# B&R Automation Studio project cnc
Automation Studio 4.3.6.57 SP; technology packages: Acp10Arnc0 5.2.1, mapp 5.2.1

## Configuration X20CP1382SM

CPU X20CP1382, AutomationRuntime G4.34, Build 4.1.2, Vc V4.34.2

### Task classes (Cpu.sw)
```
Cyclic#1 (cycle 4000 us, tolerance 0 us):
  ncsdcctrl <- Motion.Stepper.ncsdcctrl.prg
Cyclic#3:
  Cnc <- Motion.Cnc.prg
  MFunc <- Motion.MFunc.prg
Cyclic#4:
  Draw <- Visualization.Draw.prg
DataObjects: Acp10sys, Arnc0sys
NcDataObjects: CncInit <- Motion.CncInit.dob, gmcipvar <- GmcIpUserConfig.gmcipvar.dob, gmcipfun <- GmcIpUserConfig.gmcipfun.dob, gmcipfub <- GmcIpUserConfig.gmcipfub.dob, gmcipubr <- GmcIpUserConfig.gmcipubr.dob, gmcipusm <- GmcIpUserConfig.gmcipusm.dob, gmcipui <- GmcIpUserConfig.gmcipui.dob, gmcipus <- GmcIpUserConfig.gmcipus.dob, gmcipuc <- GmcIpUserConfig.gmcipuc.dob, gmcipsys <- GmcIpConfig.gmcipsys.dob, gmciplbr <- GmcIpConfig.gmciplbr.dob, gmcipcbr <- GmcIpConfig.gmcipcbr.dob, gmciplsm <- GmcIpConfig.gmciplsm.dob, gmcipcsm <- GmcIpConfig.gmcipcsm.dob, gmcipcfg <- GmcIpConfig.gmcipcfg.dob, gmcipiec <- GmcIpConfig.gmcipiec.dob, gmciplog <- GmcIpConfig.gmciplog.dob, gmcipesm <- GmcIpConfig.gmcipesm.dob, gmcipmxd <- GmcIpConfig.gmcipmxd.dob, gmcipmx <- GmcIpConfig.gmcipmx.dob, gAxisXa <- Motion.Stepper.gAxisXobj.gAxisXa.dob, gAxisXi <- Motion.Stepper.gAxisXobj.gAxisXi.dob, gAxisYa <- Motion.Stepper.gAxisYobj.gAxisYa.dob, gAxisYi <- Motion.Stepper.gAxisYobj.gAxisYi.dob, acp10etxen <- Motion.acp10etxen.dob, gAxisAa <- Motion.Stepper.gAxisAobj.gAxisAa.dob, gAxisAi <- Motion.Stepper.gAxisAobj.gAxisAi.dob, Micky <- Motion.Micky.dob
VcDataObjects: Visu <- Visualization.Visu.dob
Binaries: TCData, udbdef, arsvcreg, ashwac, Config_4, Config_3, ashwd, Config_1, User, sysconf, asfw, arconfig, iomap, Role, Config, Acp10map, acp10cfg, Arnc0map, arnc0cfg, vcclbox, vcnet, Visu02, vccpopup, vccscale, Visu01, vccddbox, Visu03, vccshape, vcpkat, vctcal, vcmgr, vcpdvnc, vccline, vccovl, vcdsint, vcctext, vccslider, vcrt, vccurl, vcxml, vcshared, vccbmp, vcchspot, vcchtml, vcpdsw, vccdt, vcdsloc, vcalarm, arial, vccalarm, vccstr, vcbclass, vcgclass, vcfntttf, vccnum, vcfile, arialbd, vccbtn, vcpfx20, Config_2, vcctrend, Visu102, Visu103, vccbar, vcpfar00
Libraries: Acp10man, Acp10par, NcGlobal, MpFile, Acp10_MC, brsystem, sys_lib, runtime, Acp10sim, MpCom, MpAxis, Arnc0man, DataObj, AsArLog, FileIO, AsArProf, AsMem, astime, MpCnc, GmcArncGrp, GmcManager, MpWebXs, AsArSdm, Acp10sdc, MpAlarmX, AsBrStr, MpBase, GmcGrpAPI, asieccon, powerlnk, areventlog, vcresman, arsvcreg, ashw, visapi
```

### Hardware
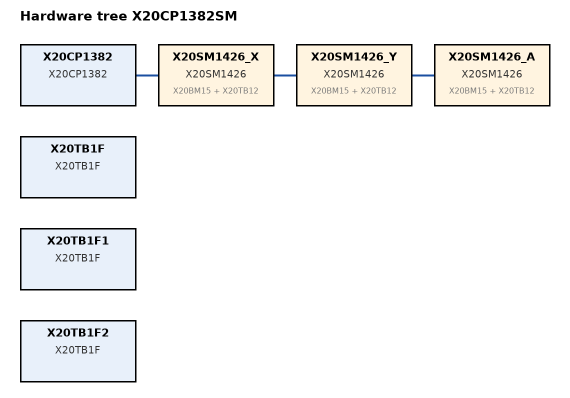
```
X20BM15 : X20BM15 v1.0.1.0  [X2X1 -> X20CP1382.IF6 (NodeNumber=1)]
X20BM15a : X20BM15 v1.0.1.0  [X2X1 -> X20BM15.X2X2 (NodeNumber=2)]
X20BM15b : X20BM15 v1.0.1.0  [X2X1 -> X20BM15a.X2X2 (NodeNumber=3)]
X20CP1382 : X20CP1382 v1.6.1.0  [X1 -> X1.SL; X2 -> X2.SL; X3 -> X3.SL]
  Module X1 (Type=X1, Virtual=true, Version=1.6.1.0)
    Connection (Connector=SS1, TargetModule=X20TB1F, TargetConnector=SS)
    Connection (Connector=SL, TargetModule=X20CP1382, TargetConnector=X1)
  Module X2 (Type=X2, Virtual=true, Version=1.6.1.0)
    Connection (Connector=SS1, TargetModule=X20TB1F1, TargetConnector=SS)
    Connection (Connector=SL, TargetModule=X20CP1382, TargetConnector=X2)
  Module X3 (Type=X3, Virtual=true, Version=1.6.1.0)
    Connection (Connector=SS1, TargetModule=X20TB1F2, TargetConnector=SS)
    Connection (Connector=SL, TargetModule=X20CP1382, TargetConnector=X3)
  Connector IF2:
    ActivateDevice = 1
    Mode = Manual
    InternetAddress = 192.168.0.1
    SubnetMask = 255.255.255.0
    InaNodeNumber = 0
    Vnc1
    VncVcObjectName1 = Visu
    VncKeyMappingFile1 = VC\PS2-Keyboard.dis
    VncRefreshRate1 = 200
  Connector IF3:
    CycleTime = 2000
  ConfigurationID = cnc_X20CP1382SM
  UserPartitionSize = 500
  Simulation = 1
  TimerDeviceType = EPLX2X
  TimerDevice = X20CP1382.IF3
  TaskClassIdleTime = 4000
  Cyclic1Duration = 4000
  Cyclic1Tolerance = 0
  FileDevice1
  FileDeviceName1 = CNC_PrgDir
  FileDevicePath1 = F:\CNC_PrgDir\
  FtpUser1
  FtpUsername1 = ich
  FtpUserPassword1 = 0jkekh+UYz/SowwWBzua0G3yXD3GBpeVHnITZJiG9J0=
  FtpUserSalt1 = 4HMg2Zqv
  FTPAccessRight1 = 0
X20SM1426_A : X20SM1426 v1.5.1.1  [SS1 -> X20TB12b.SS; SL -> X20BM15b.SL1]
  Supervision = off
  RatedCurrent = 50
  MaximumCurrent = 50
  LatchSync = Stepper latch value synchron (AB/R latch value asynchron)
  SM_SCALE_LOAD_UNITS_r1 = 36000
  SCALE_ENCOD_INCR_r1 = 51200
  CNC_r1 = on
  BothEndSwitchesAreNormallyOpen_r1 = on
  QuickStopIsNormallyOpen_r1 = on
X20SM1426_X : X20SM1426 v1.5.1.1  [SS1 -> X20TB12.SS; SL -> X20BM15.SL1]
  Supervision = off
  RatedCurrent = 50
  MaximumCurrent = 50
  LatchSync = Stepper latch value synchron (AB/R latch value asynchron)
  SM_SCALE_LOAD_UNITS_r1 = 200
  SCALE_ENCOD_INCR_r1 = 51200
  CNC_r1 = on
  BothEndSwitchesAreNormallyOpen_r1 = on
  QuickStopIsNormallyOpen_r1 = on
X20SM1426_Y : X20SM1426 v1.5.1.1  [SS1 -> X20TB12a.SS; SL -> X20BM15a.SL1]
  Supervision = off
  RatedCurrent = 50
  MaximumCurrent = 50
  LatchSync = Stepper latch value synchron (AB/R latch value asynchron)
  SM_SCALE_LOAD_UNITS_r1 = 200
  SCALE_ENCOD_INCR_r1 = 51200
  CNC_r1 = on
  BothEndSwitchesAreNormallyOpen_r1 = on
  QuickStopIsNormallyOpen_r1 = on
X20TB12 : X20TB12 v1.0.0.0
X20TB12a : X20TB12 v1.0.0.0
X20TB12b : X20TB12 v1.0.0.0
X20TB1F : X20TB1F v1.0.0.0
X20TB1F1 : X20TB1F v1.0.0.0
X20TB1F2 : X20TB1F v1.0.0.0
```

### IoMap.iom - X20CP1382/IoMap.iom
```iecst
VAR_CONFIG
	Cyclic#1.gAxisX_DrvIf.iLifeCnt AT %IB."X20SM1426_X".LifeCnt;
	Cyclic#1.gAxisX_DrvIf.iDrvOK AT %IX."X20SM1426_X".DrvOk01;
	Cyclic#1.gAxisX_DrvIf.oBoostCurrent AT %QX."X20SM1426_X".BoostCurrent01;
	Cyclic#1.gAxisX_DrvIf.oStandStillCurrent AT %QX."X20SM1426_X".StandstillCurrent01;
	Cyclic#1.gAxisX_DrvIf.oSetTime AT %QW."X20SM1426_X".SetTime01;
	Cyclic#1.gAxisX_MotorStep0 AT %QW."X20SM1426_X".Motor1Step0;
	Cyclic#1.gAxisX_DiDoIf.iLifeCntDriveEnable AT %IB."X20SM1426_X".LifeCnt;
	Cyclic#1.gAxisX_DiDoIf.iLifeCntDriveReady AT %IB."X20SM1426_X".LifeCnt;
	Cyclic#1.gAxisX_DiDoIf.iDriveReady AT %IX."X20SM1426_X".DrvOk01;
	Cyclic#1.gAxisX_DiDoIf.oDriveEnable AT %QX."X20SM1426_X".DriveEnable01;
	Cyclic#1.gAxisX_EncIf1.iLifeCnt AT %IB."X20SM1426_X".LifeCnt;
	Cyclic#1.gAxisX_EncIf1.iEncOK AT %IX."X20SM1426_X".EncOk01;
	Cyclic#1.gAxisX_EncIf1.iActPos AT %IW."X20SM1426_X".ActPos01;
	Cyclic#1.gAxisX_EncIf1.iRefPulsePos AT %IW."X20SM1426_X".RefPulsePos01;
	Cyclic#1.gAxisX_EncIf1.iRefPulseCnt AT %IB."X20SM1426_X".RefPulseCnt01;
	Cyclic#1.gAxisX_EncIf1.iActTime AT %IW."X20SM1426_X".ActTime01;
	Cyclic#1.gAxisY_DrvIf.iLifeCnt AT %IB."X20SM1426_Y".LifeCnt;
	Cyclic#1.gAxisY_DrvIf.iDrvOK AT %IX."X20SM1426_Y".DrvOk01;
	Cyclic#1.gAxisY_DrvIf.oBoostCurrent AT %QX."X20SM1426_Y".BoostCurrent01;
	Cyclic#1.gAxisY_DrvIf.oStandStillCurrent AT %QX."X20SM1426_Y".StandstillCurrent01;
	Cyclic#1.gAxisY_DrvIf.oSetTime AT %QW."X20SM1426_Y".SetTime01;
	Cyclic#1.gAxisY_MotorStep0 AT %QW."X20SM1426_Y".Motor1Step0;
	Cyclic#1.gAxisY_DiDoIf.iLifeCntDriveEnable AT %IB."X20SM1426_Y".LifeCnt;
	Cyclic#1.gAxisY_DiDoIf.iLifeCntDriveReady AT %IB."X20SM1426_Y".LifeCnt;
	Cyclic#1.gAxisY_DiDoIf.iDriveReady AT %IX."X20SM1426_Y".DrvOk01;
	Cyclic#1.gAxisY_DiDoIf.oDriveEnable AT %QX."X20SM1426_Y".DriveEnable01;
	Cyclic#1.gAxisY_EncIf1.iLifeCnt AT %IB."X20SM1426_Y".LifeCnt;
	Cyclic#1.gAxisY_EncIf1.iEncOK AT %IX."X20SM1426_Y".EncOk01;
	Cyclic#1.gAxisY_EncIf1.iActPos AT %IW."X20SM1426_Y".ActPos01;
	Cyclic#1.gAxisY_EncIf1.iRefPulsePos AT %IW."X20SM1426_Y".RefPulsePos01;
	Cyclic#1.gAxisY_EncIf1.iRefPulseCnt AT %IB."X20SM1426_Y".RefPulseCnt01;
	Cyclic#1.gAxisY_EncIf1.iActTime AT %IW."X20SM1426_Y".ActTime01;
	Cyclic#1.gAxisA_DrvIf.iLifeCnt AT %IB."X20SM1426_A".LifeCnt;
	Cyclic#1.gAxisA_DrvIf.iDrvOK AT %IX."X20SM1426_A".DrvOk01;
	Cyclic#1.gAxisA_DrvIf.oBoostCurrent AT %QX."X20SM1426_A".BoostCurrent01;
	Cyclic#1.gAxisA_DrvIf.oStandStillCurrent AT %QX."X20SM1426_A".StandstillCurrent01;
	Cyclic#1.gAxisA_DrvIf.oSetTime AT %QW."X20SM1426_A".SetTime01;
	Cyclic#1.gAxisA_MotorStep0 AT %QW."X20SM1426_A".Motor1Step0;
	Cyclic#1.gAxisA_DiDoIf.iLifeCntDriveEnable AT %IB."X20SM1426_A".LifeCnt;
	Cyclic#1.gAxisA_DiDoIf.iLifeCntDriveReady AT %IB."X20SM1426_A".LifeCnt;
	Cyclic#1.gAxisA_DiDoIf.iDriveReady AT %IX."X20SM1426_A".DrvOk01;
	Cyclic#1.gAxisA_DiDoIf.oDriveEnable AT %QX."X20SM1426_A".DriveEnable01;
	Cyclic#1.gAxisA_EncIf1.iLifeCnt AT %IB."X20SM1426_A".LifeCnt;
	Cyclic#1.gAxisA_EncIf1.iEncOK AT %IX."X20SM1426_A".EncOk01;
	Cyclic#1.gAxisA_EncIf1.iActPos AT %IW."X20SM1426_A".ActPos01;
	Cyclic#1.gAxisA_EncIf1.iRefPulsePos AT %IW."X20SM1426_A".RefPulsePos01;
	Cyclic#1.gAxisA_EncIf1.iRefPulseCnt AT %IB."X20SM1426_A".RefPulseCnt01;
	Cyclic#1.gAxisA_EncIf1.iActTime AT %IW."X20SM1426_A".ActTime01;
END_VAR
```

### Acp10cfg.ncc - X20CP1382/Motion/Acp10cfg.ncc
```
NcConfiguration (Version=3.12.1, NcSwId=Acp10)
  ACP10CF1_typ:
    cnt_nettrc_rec_drive = 1500
    bufsize_trace_upload = 1200
    tc_nc_man_task = Cyclic #1
    glob_pv_as_ncobject = Yes
    ncsys_dl_broadcast = Yes
    ncsys_dl_acp_reset = Yes
    safemc_log_err_to_ax = Yes
    network_init:
      ncsw_init_execute = Yes
      automatic_execute = No
      node_nr_warning = Yes
      net_err_before_ncact = Yes
    nettrc:
      enter_parsecrec = Yes
      enter_ncaction = Yes
      save_ring_startidx = Yes
    cam_prof_download:
      cam_dat_dl_parallel = No
      tc_cam_dl_parallel = Task class for NC Manager task
    plk_if[0]:
      if_name = IF3
      tc_CycDat_PLCopen = Task class for NC Manager task
      mc_broadcast_extdat = No
    sdc_if[0]:
      if_name = SDC_IF1
      mc_broadcast_size = 800
      mc_broadcast_extdat = No
```

### Acp10map.ncm - X20CP1382/Motion/Acp10map.ncm
```
NcMapping (NcSwId=Acp10, DisabledNodesAreHidden=False)
  NcObject gAxisX (ModuleId=X20SM1426_X, ModuleAddress=SDC_IF1.ST1, Type=ncAXIS, Channel=1, AcoposSimulation=Off, InitParameter=gAxisXi, AcoposParameter=gAxisXa, AdditionalData=CNC_Enabled="1", Disabled=FALSE, ModuleDisabled=FALSE)
  NcObject gAxisY (ModuleId=X20SM1426_Y, ModuleAddress=SDC_IF1.ST2, Type=ncAXIS, Channel=1, AcoposSimulation=Off, InitParameter=gAxisYi, AcoposParameter=gAxisYa, AdditionalData=CNC_Enabled="1", Disabled=FALSE, ModuleDisabled=FALSE)
  NcObject gAxisA (ModuleId=X20SM1426_A, ModuleAddress=SDC_IF1.ST3, Type=ncAXIS, Channel=1, AcoposSimulation=Off, InitParameter=gAxisAi, AcoposParameter=gAxisAa, AdditionalData=CNC_Enabled="1", Disabled=FALSE, ModuleDisabled=FALSE)
```

### Arnc0cfg.ncc - X20CP1382/Motion/Arnc0cfg.ncc
```
NcConfiguration (Version=3.11.0, NcSwId=Arnc0)
  ARNC0CFG_typ:
    sampling_rate = 4000
    cnt_nettrc_rec_drive = 150
    bufsize_sys_trace = 16#00005000
    enable_mp_log = Yes
    tc_nc_man_task = Cyclic #1
    bg_load = 1
    glob_pv_as_ncobject = No
```

### Arnc0map.ncm - X20CP1382/Motion/Arnc0map.ncm
```
NcMapping (NcSwId=Arnc0, DisabledNodesAreHidden=False)
  NcObject gCnc1 (Type=ncCNCSYS, Channel=1, AcoposSimulation=Off, InitParameter=CncInit, Disabled=FALSE, ModuleDisabled=FALSE)
  NcObject CNC2 (Type=ncCNCSYS, Channel=2, AcoposSimulation=Off, Disabled=TRUE, ModuleDisabled=FALSE)
  NcObject CNC3 (Type=ncCNCSYS, Channel=3, AcoposSimulation=Off, Disabled=TRUE, ModuleDisabled=FALSE)
  NcObject CNC4 (Type=ncCNCSYS, Channel=4, AcoposSimulation=Off, Disabled=TRUE, ModuleDisabled=FALSE)
  NcObject CNC5 (Type=ncCNCSYS, Channel=5, AcoposSimulation=Off, Disabled=TRUE, ModuleDisabled=FALSE)
  NcObject CNC6 (Type=ncCNCSYS, Channel=6, AcoposSimulation=Off, Disabled=TRUE, ModuleDisabled=FALSE)
  NcObject CNC7 (Type=ncCNCSYS, Channel=7, AcoposSimulation=Off, Disabled=TRUE, ModuleDisabled=FALSE)
  NcObject CNC8 (Type=ncCNCSYS, Channel=8, AcoposSimulation=Off, Disabled=TRUE, ModuleDisabled=FALSE)
  NcObject CNC9 (Type=ncCNCSYS, Channel=9, AcoposSimulation=Off, Disabled=TRUE, ModuleDisabled=FALSE)
  NcObject CNC10 (Type=ncCNCSYS, Channel=10, AcoposSimulation=Off, Disabled=TRUE, ModuleDisabled=FALSE)
  NcObject CNC11 (Type=ncCNCSYS, Channel=11, AcoposSimulation=Off, Disabled=TRUE, ModuleDisabled=FALSE)
  NcObject CNC12 (Type=ncCNCSYS, Channel=12, AcoposSimulation=Off, Disabled=TRUE, ModuleDisabled=FALSE)
  NcObject CNC13 (Type=ncCNCSYS, Channel=13, AcoposSimulation=Off, Disabled=TRUE, ModuleDisabled=FALSE)
  NcObject CNC14 (Type=ncCNCSYS, Channel=14, AcoposSimulation=Off, Disabled=TRUE, ModuleDisabled=FALSE)
  NcObject CNC15 (Type=ncCNCSYS, Channel=15, AcoposSimulation=Off, Disabled=TRUE, ModuleDisabled=FALSE)
  NcObject CNC16 (Type=ncCNCSYS, Channel=16, AcoposSimulation=Off, Disabled=TRUE, ModuleDisabled=FALSE)
  NcObject CNC17 (Type=ncCNCSYS, Channel=17, AcoposSimulation=Off, Disabled=TRUE, ModuleDisabled=FALSE)
  NcObject CNC18 (Type=ncCNCSYS, Channel=18, AcoposSimulation=Off, Disabled=TRUE, ModuleDisabled=FALSE)
  NcObject CNC19 (Type=ncCNCSYS, Channel=19, AcoposSimulation=Off, Disabled=TRUE, ModuleDisabled=FALSE)
  NcObject CNC20 (Type=ncCNCSYS, Channel=20, AcoposSimulation=Off, Disabled=TRUE, ModuleDisabled=FALSE)
  NcObject CNC21 (Type=ncCNCSYS, Channel=21, AcoposSimulation=Off, Disabled=TRUE, ModuleDisabled=FALSE)
  NcObject CNC22 (Type=ncCNCSYS, Channel=22, AcoposSimulation=Off, Disabled=TRUE, ModuleDisabled=FALSE)
  NcObject CNC23 (Type=ncCNCSYS, Channel=23, AcoposSimulation=Off, Disabled=TRUE, ModuleDisabled=FALSE)
  NcObject CNC24 (Type=ncCNCSYS, Channel=24, AcoposSimulation=Off, Disabled=TRUE, ModuleDisabled=FALSE)
```

### Config.mpaxisbasic - X20CP1382/Motion/Config.mpaxisbasic
```
Element gMpAxisY (Type=mpaxisbasic)
  AxisConfiguration = AxisWithConfiguration
    AxisName = Y
    Axis:
      BaseType = 0
      MeasurementUnit = 1
      PeriodSettings:
        Period = 0
      MovementLimits:
        VelocityPositive = 8
        VelocityNegative = 8
        Acceleration = 50
        Deceleration = 50
    Drive:
      Gearbox:
        Output = 2
      Transformation:
        ReferenceDistance = 1
      Controller:
        LoopFilters:
          [0]
          [1]
          [2]
  Alarms = MpAlarmX
Element gMpAxisX (Type=mpaxisbasic)
  AxisConfiguration = AxisWithConfiguration
    AxisName = X
    Axis:
      BaseType = 0
      MeasurementUnit = 1
      PeriodSettings:
        Period = 0
      MovementLimits:
        VelocityPositive = 8
        VelocityNegative = 8
        Acceleration = 50
        Deceleration = 50
    Drive:
      Gearbox:
        Output = 2
      Transformation:
        ReferenceDistance = 1
      Controller:
        LoopFilters:
          [0]
          [1]
          [2]
  Alarms = MpAlarmX
Element gMpAxisA (Type=mpaxisbasic)
  AxisConfiguration = AxisWithConfiguration
    AxisName = A
    Axis:
      BaseType = 1
      PeriodSettings:
        Period = 0
      MovementLimits:
        VelocityPositive = 90
        VelocityNegative = 90
        Acceleration = 100
        Deceleration = 100
    Drive:
      Controller:
        LoopFilters:
          [0]
          [1]
          [2]
  Alarms = MpAlarmX
```

### Config_4.mpcnc3axis - X20CP1382/Motion/Config_4.mpcnc3axis
```
Element gMpCnc1 (Type=mpcnc3axis)
  Linking:
    Subnodes:
      AxisX = gMpAxisX
      AxisY = gMpAxisY
      AxisZ = gMpAxisA
  Cnc:
    CncName = CNC1
  Alarms = MpAlarmX
    mapp.AlarmX.Core.Configuration:
      [0]:
        Code = 1001
      [1]:
        Code = 1002
      [2]:
        Code = 1003
      [3]:
        Code = 1004
      [4]:
        Code = 1005
      [5]:
        Code = 1006
      [6]:
        Code = 1007
```

### Config_3.mpfilemanagerui - X20CP1382/mappServices/Config_3.mpfilemanagerui
```
Element gCncFileManagerUI (Type=mpfilemanagerui)
  FileMan:
    CustomizedFileType:
      [0] = cnc
```

## Logical view

Binary libraries used (declarations not repeated): operator, runtime, astime, AsIecCon, brsystem, sys_lib, DataObj, AsArLog, FileIO, AsArProf, AsMem, AsArSdm, standard, ArEventLog, AsBrStr, visapi, MpCnc 1.65.0, GmcGrpAPI 5.02.1, GmcArncGrp 5.02.1, MpAxis 1.65.0, GmcManager 5.02.1, NcGlobal 5.02.1, MpBase, Arnc0man 5.02.1, Acp10_MC 5.02.1, Acp10man 5.02.1, Acp10par 5.02.1, Acp10sim 5.02.1, Acp10sdc 5.02.1, MpWebXs, MpFile 5.02.1, MpCom 5.02.1, MpAlarmX 5.02.1

### Motion.var
```iecst
VAR
	gAxisX : ACP10AXIS_typ;
	gAxisY : ACP10AXIS_typ;
	gAxisA : ACP10AXIS_typ;
	gCnc1 : MCAxesGroupType_Arnc := (0);
	g_positionY : LREAL;
	g_positionX : LREAL;
END_VAR
```

### Program Logical/Motion/Cnc (IEC)

#### Cyclic.st - Cyclic code
```iecst
PROGRAM _CYCLIC

	FOR n := 0 TO MAX_AXES_MINUS_ONE DO
		Axis[n].MpAxis();
	END_FOR

	FOR n := 0 TO MAX_CNC_MINUS_ONE DO
		Cnc[n].MpCnc();
		CncCyclicAction;

	END_FOR

	g_positionX := Cnc[0].MpCnc.X;
	g_positionY := Cnc[0].MpCnc.Y;

	FileHandling.fileManager();

	(* mapp logger *)
	Logger.UI();

	(* gmc logger *)
	ReadEventLogger;

	AlarmHandling.MpAlarmXCore();
	AlarmHandling.UIList();

	(* interface to visu *)
	IF NOT(Cnc[0].MpCnc.MoveProgram) THEN
		statusFlags.0 := 0;  (* stop *)
		statusFlags.1 := 0;
	ELSIF ABS(Cnc[0].MpCnc.Override) < 0.1 THEN
		statusFlags.0 := 1;  (* paused *)
		statusFlags.1 := 0;
	ELSE
		IF Cnc[0].MpCnc.Override > 0 THEN
			statusFlags.0 := 0;  (* start *)
			statusFlags.1 := 1;
		ELSE
			statusFlags.0 := 1;  (* back *)
			statusFlags.1 := 1;
		END_IF
	END_IF

	statusFlags.31 := Cnc[0].MpCnc.Error OR Axis[0].MpAxis.Error OR Axis[1].MpAxis.Error OR Axis[2].MpAxis.Error;

END_PROGRAM
```

#### Init_Exit.st - Init & Exit code
```iecst
PROGRAM _INIT

	(* Axes *)
	Axis[0].MpAxis.Axis := ADR(gAxisX);
	Axis[0].MpAxis.MpLink := ADR(gMpAxisX);

	Axis[1].MpAxis.Axis := ADR(gAxisY);
	Axis[1].MpAxis.MpLink := ADR(gMpAxisY);

	Axis[2].MpAxis.Axis := ADR(gAxisA);
	Axis[2].MpAxis.MpLink := ADR(gMpAxisA);

	FOR n := 0 TO MAX_AXES_MINUS_ONE DO
		Axis[n].MpAxisParameter.Jog.LowerLimit := -1000;
		Axis[n].MpAxisParameter.Jog.UpperLimit := 1000;
		Axis[n].MpAxisParameter.Jog.Acceleration := 20;
		Axis[n].MpAxisParameter.Jog.Deceleration := 20;
		Axis[n].MpAxisParameter.Jog.Velocity := 1;
		Axis[n].MpAxis.Parameters := ADR(Axis[n].MpAxisParameter);
		Axis[n].MpAxis.Enable := TRUE;
	END_FOR

	(* Cnc *)
	Cnc[0].MpCnc.AxesGroup := ADR(gCnc1);
	Cnc[0].MpCnc.MpLink := ADR(gMpCnc1);
	Cnc[0].MpCnc.Enable := TRUE;

	FOR n := 0 TO MAX_CNC_MINUS_ONE DO
		Cnc[0].step := W_AXES_READY;
		Cnc[0].MpCnc.Override := 100;
		Cnc[n].MpCnc.Parameters := ADR(Cnc[n].MpCncParameter);
	END_FOR

	Cnc[0].MpCncParameter.ProgramName := 'Micky';

	(* File Handling *)
	FileHandling.fileManager.MpLink := ADR(gCncFileManagerUI);
	FileHandling.fileManager.UISetup.FileListSize := 5;
	FileHandling.fileManager.UISetup.FileListScrollWindow := 1;
	FileHandling.UIConnect.DeviceList.DeviceNames[0] := 'CNC_PrgDir';
	FileHandling.fileManager.UIConnect := ADR(FileHandling.UIConnect);
	FileHandling.fileManager.Enable := TRUE;

	(* mapp Logging *)
	Logger.UI.MpLink := ADR(gMpCnc1);
	Logger.UI.Scope := mpCOM_CONFIG_SCOPE_BRANCH;
	Logger.UI.Enable := TRUE;
	Logger.UI.EntryFilter := 'Severity=ERROR';
	Logger.UI.UISetup.LoggerListSize := 1;
	Logger.UI.UISetup.LoggerScrollWindow := 1;
	Logger.UI.UIConnect := ADR(Logger.UIConnect);

	(* GMC Logging via ArEventLog *)
	Logger.eventLog.ArEventLogGetIdent.Name := 'GMC';

	(* Alarm Handling *)
	AlarmHandling.MpAlarmXCore.MpLink := ADR(gAlarmXCore);
	AlarmHandling.MpAlarmXCore.Enable := TRUE;
	AlarmHandling.UIList.MpLink := ADR(gAlarmXCore);
	AlarmHandling.UIList.Enable := TRUE;
	AlarmHandling.UIList.UISetup.AlarmListScrollWindow := 1;
	AlarmHandling.UIList.UISetup.AlarmListSize := 20;
	AlarmHandling.UIList.UIConnect := ADR(AlarmHandling.UIConnect);

END_PROGRAM

PROGRAM _EXIT
	FOR n := 0 TO MAX_CNC_MINUS_ONE DO
		Cnc[n].MpCnc( Enable := FALSE );
	END_FOR
	FOR n := 0 TO MAX_AXES_MINUS_ONE DO
		Axis[n].MpAxis( Enable := FALSE );
	END_FOR
	Logger.UI( Enable := FALSE );
	AlarmHandling.MpAlarmXCore( Enable := FALSE );
	AlarmHandling.UIList( Enable := FALSE );

	Logger.eventLog.ArEventLogGetIdent( Execute := FALSE );
END_PROGRAM
```

#### Types.typ - Local data types
```iecst
TYPE
	FileHandlingType : 	STRUCT
		fileManager : MpFileManagerUI;
		UIConnect : MpFileManagerUIConnectType;
	END_STRUCT;
	AlarmHandlingType : 	STRUCT
		MpAlarmXCore : MpAlarmXCore;
		UIConnect : MpAlarmXListUIConnectType;
		UIList : MpAlarmXListUI;
	END_STRUCT;
	EventLoggingEntryType : 	STRUCT
		dt : DATE_AND_TIME;
		TimeStamp : ArEventLogTimeStampType;
		RecordID : ArEventLogRecordIDType;
		EventID : DINT;
		text : STRING[255];
	END_STRUCT;
	EventLoggingType : 	STRUCT
		step : USINT;
		index : INT;
		maxIndex : INT;
		entries : ARRAY[0..19]OF EventLoggingEntryType;
		ArEventLogGetIdent : ArEventLogGetIdent;
		ArEventLogGetLatestRecordID : ArEventLogGetLatestRecordID;
		ArEventLogGetPreviousRecordID : ArEventLogGetPreviousRecordID;
		ArEventLogRead : ArEventLogRead;
		ArEventLogReadAddData : ArEventLogReadAddData;
	END_STRUCT;
	LoggingType : 	STRUCT
		UIConnect : MpComLoggerUIConnectType;
		UI : MpComLoggerUI;
		eventLog : EventLoggingType;
	END_STRUCT;
	CncType : 	STRUCT
		MpCnc : MpCnc3Axis;
		MpCncParameter : MpCnc3AxisParType;
		step : UINT;
	END_STRUCT;
	AxisType : 	STRUCT
		MpAxis : MpAxisBasic;
		MpAxisParameter : MpAxisBasicParType;
	END_STRUCT;
END_TYPE
```

#### Variables.var - Local variables
```iecst
VAR
	Logger : LoggingType;
	FileHandling : FileHandlingType;
	AlarmHandling : AlarmHandlingType;
	Cnc : ARRAY[0..MAX_CNC_MINUS_ONE] OF CncType;
	n : UINT;
END_VAR
VAR CONSTANT
	MAX_AXES_MINUS_ONE : USINT := MAX_AXES-1;
	MAX_AXES : USINT := 3;
	MAX_CNC : USINT := 1;
	MAX_CNC_MINUS_ONE : USINT := MAX_CNC-1;
END_VAR
VAR
	Axis : ARRAY[0..MAX_AXES_MINUS_ONE] OF AxisType;
END_VAR
VAR CONSTANT
	W_AXES_READY : UINT := 0;
	W_POWER_ON : UINT := 10;
	W_AXES_HOMED : UINT := 20;
	W_COMMAND : UINT := 100;
END_VAR
VAR
	cnc : REFERENCE TO CncType;
	statusFlags : UDINT;
END_VAR
```

#### CncCyclicAction.st
```iecst
ACTION CncCyclicAction:

	cnc ACCESS ADR(Cnc[n]);

	CASE Cnc[n].step OF
		W_AXES_READY:
		IF cnc.MpCnc.Info.AxesReady THEN
			//cnc.MpCnc.Power := TRUE;
			cnc.step := W_POWER_ON;
		END_IF

		W_POWER_ON:
		IF cnc.MpCnc.PowerOn THEN
			//cnc.MpCnc.Home := TRUE;
			cnc.step := W_AXES_HOMED;
		END_IF

		W_AXES_HOMED:
		IF cnc.MpCnc.IsHomed THEN
			cnc.step := W_COMMAND;
		END_IF

		W_COMMAND:
		IF cnc.MpCnc.Stop AND cnc.MpCnc.Stopped THEN
			cnc.MpCnc.Stop := FALSE;
		END_IF
		IF cnc.MpCnc.IsHomed THEN
			cnc.MpCnc.Home := FALSE;
		END_IF
		IF cnc.MpCnc.ErrorReset AND cnc.MpCnc.Error = FALSE THEN
			cnc.MpCnc.ErrorReset := FALSE;
		END_IF

	END_CASE

END_ACTION
```

#### ReadEventLogger.st
```iecst
ACTION ReadEventLogger:

	CASE Logger.eventLog.step OF
		0: (* wait for start *)

		10: (* wait for ..GetIdent *)
		Logger.eventLog.ArEventLogGetIdent( Execute := TRUE );
		IF Logger.eventLog.ArEventLogGetIdent.Done THEN
			Logger.eventLog.ArEventLogGetLatestRecordID.Ident := Logger.eventLog.ArEventLogGetIdent.Ident;
			Logger.eventLog.ArEventLogGetPreviousRecordID.Ident := Logger.eventLog.ArEventLogGetIdent.Ident;
			Logger.eventLog.ArEventLogRead.Ident := Logger.eventLog.ArEventLogGetIdent.Ident;
			Logger.eventLog.ArEventLogReadAddData.Ident := Logger.eventLog.ArEventLogGetIdent.Ident;
			Logger.eventLog.maxIndex := SIZEOF(Logger.eventLog.entries)/SIZEOF(Logger.eventLog.entries[0])-1;
			brsmemset( ADR(Logger.eventLog.entries), 0, SIZEOF(Logger.eventLog.entries) );
			Logger.eventLog.ArEventLogGetIdent( Execute := FALSE );
			Logger.eventLog.index := 1;
			Logger.eventLog.step := 20;
		END_IF

		20: (* start reading latest entry *)
		Logger.eventLog.ArEventLogGetLatestRecordID( Execute := TRUE );
		IF Logger.eventLog.ArEventLogGetLatestRecordID.Done THEN
			Logger.eventLog.entries[0].RecordID := Logger.eventLog.ArEventLogGetLatestRecordID.RecordID;
			Logger.eventLog.ArEventLogGetLatestRecordID( Execute := FALSE );
			Logger.eventLog.step := 30;
		END_IF

		30: (* read previous entry *)
		IF Logger.eventLog.index <= Logger.eventLog.maxIndex THEN
			Logger.eventLog.ArEventLogGetPreviousRecordID.RecordID := Logger.eventLog.entries[Logger.eventLog.index-1].RecordID;
			Logger.eventLog.ArEventLogGetPreviousRecordID( Execute := TRUE );
			IF Logger.eventLog.ArEventLogGetPreviousRecordID.Done THEN
				Logger.eventLog.entries[Logger.eventLog.index].RecordID := Logger.eventLog.ArEventLogGetPreviousRecordID.PrevRecordID;
				Logger.eventLog.index := Logger.eventLog.index + 1;
			ELSIF Logger.eventLog.ArEventLogGetPreviousRecordID.Error AND Logger.eventLog.ArEventLogGetPreviousRecordID.StatusID = arEVENTLOG_ERR_RECORDID_INVALID THEN  (* end of logger *)
				Logger.eventLog.index := Logger.eventLog.index - 1;
				Logger.eventLog.step := 40;
			END_IF
			Logger.eventLog.ArEventLogGetPreviousRecordID( Execute := FALSE );
		ELSE
			Logger.eventLog.index := Logger.eventLog.index - 1;
			Logger.eventLog.step := 40;
		END_IF

		40: (* read entry information *)
		IF Logger.eventLog.index >= 0 THEN
			Logger.eventLog.ArEventLogRead( RecordID := Logger.eventLog.entries[Logger.eventLog.index].RecordID, Execute := TRUE );
			Logger.eventLog.ArEventLogReadAddData( Execute := TRUE, RecordID := Logger.eventLog.entries[Logger.eventLog.index].RecordID,
													AddData := ADR(Logger.eventLog.entries[Logger.eventLog.index].text),
													BytesToRead := SIZEOF(Logger.eventLog.entries[Logger.eventLog.index].text) );

			IF Logger.eventLog.ArEventLogRead.Done AND Logger.eventLog.ArEventLogReadAddData.Done THEN
				Logger.eventLog.entries[Logger.eventLog.index].TimeStamp := Logger.eventLog.ArEventLogRead.TimeStamp;
				Logger.eventLog.index := Logger.eventLog.index - 1;
				Logger.eventLog.ArEventLogRead( Execute := FALSE );
				Logger.eventLog.ArEventLogReadAddData( Execute := FALSE );
			END_IF
		ELSE
			Logger.eventLog.step := 0;
		END_IF

	END_CASE

	Logger.eventLog.ArEventLogRead();

END_ACTION
```

### Data object Logical/Motion/CncInit (Cns)

- CncInit.cns (not shown)

### Program Logical/Motion/MFunc (IEC)

#### Cyclic.st - Cyclic code
```iecst
PROGRAM _CYCLIC
	MC_BR_MFunction_0(AxesGroup := ADR(gCnc1), Enable := TRUE, MFunction := 7);
	IF MC_BR_MFunction_0.Value THEN
		MC_BR_MFunction_0.Reset := TRUE;
	ELSE
		MC_BR_MFunction_0.Reset := FALSE;
	END_IF

	MC_BR_MFunction_1(AxesGroup := ADR(gCnc1), Enable := TRUE, MFunction := 8);
	IF MC_BR_MFunction_1.Value THEN
		MC_BR_MFunction_1.Reset := TRUE;
	ELSE
		MC_BR_MFunction_1.Reset := FALSE;
	END_IF

END_PROGRAM
```

#### Init.st - Init code
```iecst
PROGRAM _INIT

END_PROGRAM
```

#### Variables.var - Local variables
```iecst
VAR
	MC_BR_MFunction_0 : MC_BR_MFunction;
	MC_BR_MFunction_1 : MC_BR_MFunction;
END_VAR
```

### Stepper.var
```iecst
VAR
	gAxisX_HW : SdcHwCfg_typ := (0);
	gAxisX_DrvIf : SdcDrvIf16_typ := (0);
	gAxisX_EncIf1 : SdcEncIf16_typ := (0);
	gAxisX_DiDoIf : SdcDiDoIf_typ := (0);
	gAxisX_MotorStep0 : INT := (0);
	gAxisY_HW : SdcHwCfg_typ := (0);
	gAxisY_DrvIf : SdcDrvIf16_typ := (0);
	gAxisY_EncIf1 : SdcEncIf16_typ := (0);
	gAxisY_DiDoIf : SdcDiDoIf_typ := (0);
	gAxisY_MotorStep0 : INT := (0);
	gAxisA_HW : SdcHwCfg_typ := (0);
	gAxisA_DrvIf : SdcDrvIf16_typ := (0);
	gAxisA_EncIf1 : SdcEncIf16_typ := (0);
	gAxisA_DiDoIf : SdcDiDoIf_typ := (0);
	gAxisA_MotorStep0 : INT := (0);
END_VAR
```

### Program Logical/Motion/Stepper/ncsdcctrl (IEC)

#### ncsdcctrl.var
```iecst
VAR
	gAxisY_oSetPosOld : INT := 0;
	gAxisX_oSetPosOld : INT := 0;
	gAxisA_oSetPosOld : INT := 0;
END_VAR
```

#### ncsdcctrlCyclic.st
```iecst
PROGRAM _CYCLIC

(* ### BEGIN gAxisX ### *)

(* life counter emulation of digital inputs *)
       gAxisX_DiDoIf.iLifeCntReference := gAxisX_DiDoIf.iLifeCntReference + 1;
       gAxisX_DiDoIf.iLifeCntNegHwEnd  := gAxisX_DiDoIf.iLifeCntNegHwEnd  + 1;
       gAxisX_DiDoIf.iLifeCntPosHwEnd  := gAxisX_DiDoIf.iLifeCntPosHwEnd  + 1;

(* default function model of ACOPOSmicro: convert absolute steps to delta steps - overflow save delta calculation *)
       gAxisX_MotorStep0 := gAxisX_DrvIf.oSetPos - gAxisX_oSetPosOld;
       gAxisX_oSetPosOld := gAxisX_DrvIf.oSetPos;

(* ### END gAxisX ### *)

(* ### BEGIN gAxisY ### *)

(* life counter emulation of digital inputs *)
       gAxisY_DiDoIf.iLifeCntReference := gAxisY_DiDoIf.iLifeCntReference + 1;
       gAxisY_DiDoIf.iLifeCntNegHwEnd  := gAxisY_DiDoIf.iLifeCntNegHwEnd  + 1;
       gAxisY_DiDoIf.iLifeCntPosHwEnd  := gAxisY_DiDoIf.iLifeCntPosHwEnd  + 1;

(* default function model of ACOPOSmicro: convert absolute steps to delta steps - overflow save delta calculation *)
       gAxisY_MotorStep0 := gAxisY_DrvIf.oSetPos - gAxisY_oSetPosOld;
       gAxisY_oSetPosOld := gAxisY_DrvIf.oSetPos;

(* ### END gAxisY ### *)

(* ### BEGIN gAxisA ### *)

(* life counter emulation of digital inputs *)
       gAxisA_DiDoIf.iLifeCntReference := gAxisA_DiDoIf.iLifeCntReference + 1;
       gAxisA_DiDoIf.iLifeCntNegHwEnd  := gAxisA_DiDoIf.iLifeCntNegHwEnd  + 1;
       gAxisA_DiDoIf.iLifeCntPosHwEnd  := gAxisA_DiDoIf.iLifeCntPosHwEnd  + 1;

(* default function model of ACOPOSmicro: convert absolute steps to delta steps - overflow save delta calculation *)
       gAxisA_MotorStep0 := gAxisA_DrvIf.oSetPos - gAxisA_oSetPosOld;
       gAxisA_oSetPosOld := gAxisA_DrvIf.oSetPos;

(* ### END gAxisA ### *)

END_PROGRAM
```

#### ncsdcctrlInit.st
```iecst
PROGRAM _INIT

(* ### BEGIN gAxisX ### *)

(* initialize general interfaces *)
       gAxisX.size := gAxisX.size;
       gAxisX_HW.DrvIf_Typ := ncSDC_DRVSM16;
       brsstrcpy( ADR(gAxisX_HW.DrvIf_Name[0]), ADR('gAxisX_DrvIf') );
       gAxisX_HW.DiDoIf_Typ := ncSDC_DIDO;
       brsstrcpy( ADR(gAxisX_HW.DiDoIf_Name[0]), ADR('gAxisX_DiDoIf') );
       gAxisX_HW.EncIf1_Typ := ncSDC_ENC16;
       brsstrcpy( ADR(gAxisX_HW.EncIf1_Name[0]), ADR('gAxisX_EncIf1') );
       gAxisX_EncIf1.iLifeCnt := gAxisX_EncIf1.iLifeCnt;

(* initialize old-value for delta step calculation *)
       gAxisX_oSetPosOld := gAxisX_DrvIf.oSetPos;

(* ### END gAxisX ### *)

(* ### BEGIN gAxisY ### *)

(* initialize general interfaces *)
       gAxisY.size := gAxisY.size;
       gAxisY_HW.DrvIf_Typ := ncSDC_DRVSM16;
       brsstrcpy( ADR(gAxisY_HW.DrvIf_Name[0]), ADR('gAxisY_DrvIf') );
       gAxisY_HW.DiDoIf_Typ := ncSDC_DIDO;
       brsstrcpy( ADR(gAxisY_HW.DiDoIf_Name[0]), ADR('gAxisY_DiDoIf') );
       gAxisY_HW.EncIf1_Typ := ncSDC_ENC16;
       brsstrcpy( ADR(gAxisY_HW.EncIf1_Name[0]), ADR('gAxisY_EncIf1') );
       gAxisY_EncIf1.iLifeCnt := gAxisY_EncIf1.iLifeCnt;

(* initialize old-value for delta step calculation *)
       gAxisY_oSetPosOld := gAxisY_DrvIf.oSetPos;

(* ### END gAxisY ### *)

(* ### BEGIN gAxisA ### *)

(* initialize general interfaces *)
       gAxisA.size := gAxisA.size;
       gAxisA_HW.DrvIf_Typ := ncSDC_DRVSM16;
       brsstrcpy( ADR(gAxisA_HW.DrvIf_Name[0]), ADR('gAxisA_DrvIf') );
       gAxisA_HW.DiDoIf_Typ := ncSDC_DIDO;
       brsstrcpy( ADR(gAxisA_HW.DiDoIf_Name[0]), ADR('gAxisA_DiDoIf') );
       gAxisA_HW.EncIf1_Typ := ncSDC_ENC16;
       brsstrcpy( ADR(gAxisA_HW.EncIf1_Name[0]), ADR('gAxisA_EncIf1') );
       gAxisA_EncIf1.iLifeCnt := gAxisA_EncIf1.iLifeCnt;

(* initialize old-value for delta step calculation *)
       gAxisA_oSetPosOld := gAxisA_DrvIf.oSetPos;

(* ### END gAxisA ### *)

END_PROGRAM
```

### Package Logical/Motion/Stepper/gAxisXobj - gAxisXobj

- Data object Logical/Motion/Stepper/gAxisXobj/gAxisXa (Apt) (no source held here)

### Data object Logical/Motion/Stepper/gAxisXobj/gAxisXi (Ax)

#### gAxisXi.ax
```
InitParameter (Version=3.13.1, NcSwId=ACP10)
  ACP10AXIS_typ:
    dig_in:
      level:
        reference = ncACTIV_HI
        pos_hw_end = ncACTIV_HI
        neg_hw_end = ncACTIV_HI
        trigger1 = ncACTIV_HI
        trigger2 = ncACTIV_HI
    encoder_if:
      parameter:
        count_dir = ncSTANDARD
        scaling:
          load:
            units = 200
            rev_motor = 1
    limit:
      parameter:
        v_pos = 800.0
        v_neg = 800.0
        a1_pos = 5000.0
        a2_pos = 5000.0
        a1_neg = 5000.0
        a2_neg = 5000.0
        t_jolt = 0.0
        t_in_pos = 0.0
        pos_sw_end = 838860700
        neg_sw_end = -838860800
        ds_warning = 200.0
        ds_stop = 200.0
        a_stop = 1.0E+30
        dv_stop = 0.0
        dv_stop_mode = ncOFF
    controller:
      mode = ncPOSITION
      position:
        kv = 50.0
        tn = 0.0
        t_predict = 0.0004
        t_total = 0.0004
        p_max = 1.0E+30
        i_max = 1.0E+30
      speed:
        kv = 2.0
        tn = 0.0
        t_filter = 0.0
        isq_filter1:
          type = ncOFF
          a0 = 0.0
          a1 = 0.0
          b0 = 0.0
          b1 = 0.0
          b2 = 0.0
          c0_par_id = 0
          c1_par_id = 0
        isq_filter2:
          type = ncOFF
          a0 = 0.0
          a1 = 0.0
          b0 = 0.0
          b1 = 0.0
          b2 = 0.0
          c0_par_id = 0
          c1_par_id = 0
        isq_filter3:
          type = ncOFF
          a0 = 0.0
          a1 = 0.0
          b0 = 0.0
          b1 = 0.0
          b2 = 0.0
          c0_par_id = 0
          c1_par_id = 0
      uf:
        type = ncLINEAR
        auto_config = ncMOTOR_PAR
        u0 = 0.0
        un = 0.0
        fn = 50.0
        k_f_slip = 0.0
      ff:
        torque_load = 0.0
        torque_pos = 0.0
        torque_neg = 0.0
        kv_torque = 0.0
        inertia = 0.0
        t_filter_a = 0.0
    move:
      stop:
        parameter[0]:
          decel_ramp = ncA_LIMIT
          controller = ncON
        parameter[1]:
          decel_ramp = ncA_LIMIT
          controller = ncON
        parameter[2]:
          decel_ramp = ncA_LIMIT
          controller = ncON
        parameter[3]:
          decel_ramp = ncA_LIMIT
          controller = ncON
        quickstop:
          decel_ramp = ncA_LIMIT
        drive_error:
          decel_ramp = ncA_LIMIT
      homing:
        parameter:
          s = 0
          v_switch = 5000.0
          v_trigger = 500.0
          a = 50000.0
          mode = ncDIRECT
          edge_sw = ncPOSITIVE
          start_dir = ncPOSITIVE
          trigg_dir = ncPOSITIVE
          ref_pulse = ncOFF
          fix_dir = ncOFF
          tr_s_block = 0.0
          torque_lim = 0.0
          ds_block = 0.0
          ds_stop = 0.0
      basis:
        parameter:
          v_pos = 800.0
          v_neg = 800.0
          a1_pos = 5000.0
          a2_pos = 5000.0
          a1_neg = 5000.0
          a2_neg = 5000.0
    message:
      text:
        parameter:
          format = ncBREAK + ncZERO
          columns = 80
          data_modul = acp10etxen
```

### Package Logical/Motion/Stepper/gAxisYobj - gAxisYobj

### Data object Logical/Motion/Stepper/gAxisYobj/gAxisYa (Apt)

#### gAxisYa.apt
```
AcoposParameterTable:
  Root Parameters:
    64232 = 51200 (Name=SM_SCALE_STEP, Disabled=FALSE)
    64233 = 200 (Name=SM_SCALE_LOAD_UNITS, Disabled=FALSE)
    64234 = 1 (Name=SM_SCALE_LOAD_MOTREV, Disabled=FALSE)
    109 = 51200 (Name=SCALE_ENCOD_INCR, Disabled=FALSE)
    230 = PCTRL_S_SET (Name=PCTRL_S_ACT_PARID)  // CTRL Position controller: Actual encoder position parameter ID
```

### Data object Logical/Motion/Stepper/gAxisYobj/gAxisYi (Ax)

#### gAxisYi.ax
```
InitParameter (Version=3.13.1, NcSwId=ACP10)
  ACP10AXIS_typ:
    dig_in:
      level:
        reference = ncACTIV_HI
        pos_hw_end = ncACTIV_HI
        neg_hw_end = ncACTIV_HI
        trigger1 = ncACTIV_HI
        trigger2 = ncACTIV_HI
    encoder_if:
      parameter:
        count_dir = ncSTANDARD
        scaling:
          load:
            units = 200
            rev_motor = 1
    limit:
      parameter:
        v_pos = 100000.0
        v_neg = 100000.0
        a1_pos = 500000.0
        a2_pos = 500000.0
        a1_neg = 500000.0
        a2_neg = 500000.0
        t_jolt = 0.0
        t_in_pos = 0.0
        pos_sw_end = 838860700
        neg_sw_end = -838860800
        ds_warning = 200.0
        ds_stop = 200.0
        a_stop = 1.0E+30
        dv_stop = 0.0
        dv_stop_mode = ncOFF
    controller:
      mode = ncPOSITION
      position:
        kv = 50.0
        tn = 0.0
        t_predict = 0.0004
        t_total = 0.0004
        p_max = 1.0E+30
        i_max = 1.0E+30
      speed:
        kv = 2.0
        tn = 0.0
        t_filter = 0.0
        isq_filter1:
          type = ncOFF
          a0 = 0.0
          a1 = 0.0
          b0 = 0.0
          b1 = 0.0
          b2 = 0.0
          c0_par_id = 0
          c1_par_id = 0
        isq_filter2:
          type = ncOFF
          a0 = 0.0
          a1 = 0.0
          b0 = 0.0
          b1 = 0.0
          b2 = 0.0
          c0_par_id = 0
          c1_par_id = 0
        isq_filter3:
          type = ncOFF
          a0 = 0.0
          a1 = 0.0
          b0 = 0.0
          b1 = 0.0
          b2 = 0.0
          c0_par_id = 0
          c1_par_id = 0
      uf:
        type = ncLINEAR
        auto_config = ncMOTOR_PAR
        u0 = 0.0
        un = 0.0
        fn = 50.0
        k_f_slip = 0.0
      ff:
        torque_load = 0.0
        torque_pos = 0.0
        torque_neg = 0.0
        kv_torque = 0.0
        inertia = 0.0
        t_filter_a = 0.0
    move:
      stop:
        parameter[0]:
          decel_ramp = ncA_LIMIT
          controller = ncON
        parameter[1]:
          decel_ramp = ncA_LIMIT
          controller = ncON
        parameter[2]:
          decel_ramp = ncA_LIMIT
          controller = ncON
        parameter[3]:
          decel_ramp = ncA_LIMIT
          controller = ncON
        quickstop:
          decel_ramp = ncA_LIMIT
        drive_error:
          decel_ramp = ncA_LIMIT
      homing:
        parameter:
          s = 0
          v_switch = 5000.0
          v_trigger = 500.0
          a = 50000.0
          mode = ncDIRECT
          edge_sw = ncPOSITIVE
          start_dir = ncPOSITIVE
          trigg_dir = ncPOSITIVE
          ref_pulse = ncOFF
          fix_dir = ncOFF
          tr_s_block = 0.0
          torque_lim = 0.0
          ds_block = 0.0
          ds_stop = 0.0
      basis:
        parameter:
          v_pos = 10000.0
          v_neg = 10000.0
          a1_pos = 20000.0
          a2_pos = 20000.0
          a1_neg = 20000.0
          a2_neg = 20000.0
    message:
      text:
        parameter:
          format = ncBREAK + ncZERO
          columns = 80
          data_modul = acp10etxen
```

### Package Logical/Motion/Stepper/gAxisAobj - gAxisYobj

### Data object Logical/Motion/Stepper/gAxisAobj/gAxisAa (Apt)

#### gAxisAa.apt
```
AcoposParameterTable:
  Root Parameters:
    64232 = 51200 (Name=SM_SCALE_STEP, Disabled=FALSE)
    64233 = 36000 (Name=SM_SCALE_LOAD_UNITS, Disabled=FALSE)
    64234 = 1 (Name=SM_SCALE_LOAD_MOTREV, Disabled=FALSE)
    109 = 51200 (Name=SCALE_ENCOD_INCR, Disabled=FALSE)
    230 = PCTRL_S_SET (Name=PCTRL_S_ACT_PARID)  // CTRL Position controller: Actual encoder position parameter ID
```

### Data object Logical/Motion/Stepper/gAxisAobj/gAxisAi (Ax)

#### gAxisAi.ax
```
InitParameter (Version=3.13.1, NcSwId=ACP10)
  ACP10AXIS_typ:
    dig_in:
      level:
        reference = ncACTIV_HI
        pos_hw_end = ncACTIV_HI
        neg_hw_end = ncACTIV_HI
        trigger1 = ncACTIV_HI
        trigger2 = ncACTIV_HI
    encoder_if:
      parameter:
        count_dir = ncSTANDARD
        scaling:
          load:
            units = 36000
            rev_motor = 1
    limit:
      parameter:
        v_pos = 9000.0
        v_neg = 9000.0
        a1_pos = 10000.0
        a2_pos = 10000.0
        a1_neg = 10000.0
        a2_neg = 10000.0
        t_jolt = 0.0
        t_in_pos = 0.0
        pos_sw_end = 838860700
        neg_sw_end = -838860800
        ds_warning = 200.0
        ds_stop = 200.0
        a_stop = 1.0E+30
        dv_stop = 0.0
        dv_stop_mode = ncOFF
    controller:
      mode = ncPOSITION
      position:
        kv = 50.0
        tn = 0.0
        t_predict = 0.0004
        t_total = 0.0004
        p_max = 1.0E+30
        i_max = 1.0E+30
      speed:
        kv = 2.0
        tn = 0.0
        t_filter = 0.0
        isq_filter1:
          type = ncOFF
          a0 = 0.0
          a1 = 0.0
          b0 = 0.0
          b1 = 0.0
          b2 = 0.0
          c0_par_id = 0
          c1_par_id = 0
        isq_filter2:
          type = ncOFF
          a0 = 0.0
          a1 = 0.0
          b0 = 0.0
          b1 = 0.0
          b2 = 0.0
          c0_par_id = 0
          c1_par_id = 0
        isq_filter3:
          type = ncOFF
          a0 = 0.0
          a1 = 0.0
          b0 = 0.0
          b1 = 0.0
          b2 = 0.0
          c0_par_id = 0
          c1_par_id = 0
      uf:
        type = ncLINEAR
        auto_config = ncMOTOR_PAR
        u0 = 0.0
        un = 0.0
        fn = 50.0
        k_f_slip = 0.0
      ff:
        torque_load = 0.0
        torque_pos = 0.0
        torque_neg = 0.0
        kv_torque = 0.0
        inertia = 0.0
        t_filter_a = 0.0
    move:
      stop:
        parameter[0]:
          decel_ramp = ncA_LIMIT
          controller = ncON
        parameter[1]:
          decel_ramp = ncA_LIMIT
          controller = ncON
        parameter[2]:
          decel_ramp = ncA_LIMIT
          controller = ncON
        parameter[3]:
          decel_ramp = ncA_LIMIT
          controller = ncON
        quickstop:
          decel_ramp = ncA_LIMIT
        drive_error:
          decel_ramp = ncA_LIMIT
      homing:
        parameter:
          s = 0
          v_switch = 5000.0
          v_trigger = 500.0
          a = 50000.0
          mode = ncDIRECT
          edge_sw = ncPOSITIVE
          start_dir = ncPOSITIVE
          trigg_dir = ncPOSITIVE
          ref_pulse = ncOFF
          fix_dir = ncOFF
          tr_s_block = 0.0
          torque_lim = 0.0
          ds_block = 0.0
          ds_stop = 0.0
      basis:
        parameter:
          v_pos = 9000.0
          v_neg = 9000.0
          a1_pos = 10000.0
          a2_pos = 10000.0
          a1_neg = 10000.0
          a2_neg = 10000.0
    message:
      text:
        parameter:
          format = ncBREAK + ncZERO
          columns = 80
          data_modul = acp10etxen
```

### Data object Logical/Motion/Micky (Cnc)

#### CncProg.cnc - CNC program (G-Code)
```
N01 %1
N10 G90 F20.0
N20 G01 X0.7677 Y0.6822
N30 X0.9831 Y0.6761
N40 X1.1227 Y0.7342
N50 X1.1212 Y0.7443
N60 X1.1212 Y0.7454 M7
N70 G03 X0.9696 Y0.9818 I-0.4585 J-0.1273
N80 G02 X0.8911 Y1.0880 I0.2197 J0.2446
N90 G02 X0.8375 Y1.2438 I0.6011 J0.2939
N100 G02 X0.8346 Y1.2688 I0.1353 J0.0279
N110 G01 X0.8497 Y1.2685 M8
N120 G03 X0.8553 Y1.2335 I0.1476 J0.0057
N130 G03 X0.8719 Y1.2052 I0.0880 J0.0326
N140 G03 X0.8971 Y1.1859 I0.0580 J0.0495
N150 G03 X0.9241 Y1.1803 I0.0246 J0.0517
N160 G03 X0.9505 Y1.1880 I-0.0023 J0.0572
N170 G03 X0.9740 Y1.2094 I-0.0383 J0.0659
N180 G03 X0.9883 Y1.2389 I-0.0761 J0.0549
N190 G03 X0.9926 Y1.2734 I-0.1125 J0.0316
N200 G01 X1.0607 Y1.2719
N210 G03 X1.0607 Y1.2671 I0.1480 J-0.0030
N220 G03 X1.0671 Y1.2256 I0.1480 J0.0018
N230 G03 X1.0833 Y1.1932 I0.1053 J0.0322
N240 G03 X1.1091 Y1.1701 I0.0664 J0.0481
N250 G03 X1.1361 Y1.1631 I0.0263 J0.0462
N260 G03 X1.1629 Y1.1708 I-0.0006 J0.0532
N270 G03 X1.1881 Y1.1945 I-0.0423 J0.0702
N280 G03 X1.2034 Y1.2273 I-0.0907 J0.0624
N290 G03 X1.2089 Y1.2689 I-0.1426 J0.0398
N300 G03 X1.2024 Y1.3104 I-0.1480 J-0.0018
N310 G03 X1.1863 Y1.3428 I-0.1053 J-0.0322
N320 G03 X1.1605 Y1.3659 I-0.0664 J-0.0481
N330 G03 X1.1335 Y1.3729 I-0.0263 J-0.0462
N340 G03 X1.1067 Y1.3653 I0.0006 J-0.0532
N350 G03 X1.0815 Y1.3416 I0.0423 J-0.0702
N360 G03 X1.0661 Y1.3087 I0.0907 J-0.0624
N370 G03 X1.0607 Y1.2733 I0.1426 J-0.0398
N380 G01 X0.9925 Y1.2753
N390 G03 X0.9853 Y1.3111 I-0.1168 J-0.0048
N400 G03 X0.9687 Y1.3394 I-0.0880 J-0.0326
N410 G03 X0.9435 Y1.3588 I-0.0580 J-0.0495
N420 G03 X0.9166 Y1.3643 I-0.0246 J-0.0517
N430 G03 X0.8901 Y1.3566 I0.0023 J-0.0572
N440 G03 X0.8666 Y1.3353 I0.0383 J-0.0659
N450 G03 X0.8549 Y1.3134 I0.0761 J-0.0549
N460 G03 X0.8497 Y1.2694 I0.1424 J-0.0392
N470 G01 X0.8346 Y1.2696
N480 G02 X0.8346 Y1.2713 I0.1381 J0.0021
N490 G01 X0.8346 Y1.2723
N500 G02 X0.8407 Y1.3121 I0.1381 J-0.0006
N510 G02 X0.8787 Y1.4182 I0.2987 J-0.0474
N520 G03 X1.4696 Y1.4545 I-4.7172 J81.4981
N530 G03 X0.8787 Y1.4182 I1.0411 J-21.7444
N540 G02 X1.1820 Y1.6496 I0.7467 J-0.6641
N550 G03 X1.6735 Y2.0027 I-0.0633 J0.6066
N560 G03 X1.5988 Y2.0149 I-0.0733 J-0.2142
N570 G02 X1.7552 Y1.9646 I-0.0036 J-0.2791
N580 G03 X1.6748 Y1.9984 I-0.1233 J-0.1804
N590 G02 X1.5755 Y1.8424 I-0.4646 J0.1861
N600 G02 X1.3183 Y1.6737 I-0.1453 J-0.0589
N610 G02 X1.0348 Y1.6574 I-0.1689 J0.4635
N620 G02 X0.8494 Y1.7047 I0.1512 J0.9805
N630 G02 X0.7192 Y1.9635 I0.0903 J0.2077
N640 G02 X0.8484 Y2.0909 I0.0469 J0.0817
N650 G02 X1.1666 Y1.9272 I-0.1851 J-0.7508
N660 G02 X1.0238 Y2.0242 I8.4233 J12.5522
N670 G02 X1.0395 Y2.0246 I0.0159 J-0.3383
N680 G01 X1.0365 Y2.0370
N690 G02 X1.0193 Y2.0588 I0.0445 J0.0526
N700 G02 X1.0092 Y2.0873 I0.1122 J0.0561
N710 G02 X1.0042 Y2.1260 I0.2037 J0.0459
N720 G02 X1.0065 Y2.1649 I0.2087 J0.0072
N730 G02 X1.0147 Y2.1940 I0.1240 J-0.0191
N740 G02 X1.0303 Y2.2170 I0.0636 J-0.0265
N750 G02 X1.0446 Y2.2231 I0.0151 J-0.0155
N760 G02 X1.0593 Y2.2180 I0.0007 J-0.0216
N770 G02 X1.0765 Y2.1962 I-0.0445 J-0.0526
N780 G02 X1.0866 Y2.1677 I-0.1122 J-0.0561
N790 G02 X1.0916 Y2.1290 I-0.2037 J-0.0459
N800 G02 X1.0893 Y2.0901 I-0.2087 J-0.0072
N810 G02 X1.0811 Y2.0610 I-0.1240 J0.0191
N820 G02 X1.0655 Y2.0380 I-0.0636 J0.0265
N830 G01 X1.0627 Y2.0238
N840 G02 X1.2575 Y1.9454 I-0.0229 J-0.3379
N850 G03 X1.2197 Y1.9731 I-0.3137 J-0.3870
N860 G01 X1.2064 Y1.9850
N870 G02 X1.1893 Y2.0133 I0.0591 J0.0548
N880 G02 X1.1820 Y2.0484 I0.1335 J0.0465
N890 G02 X1.1828 Y2.0941 I0.2292 J0.0185
N900 G02 X1.1927 Y2.1387 I0.2283 J-0.0272
N910 G02 X1.2081 Y2.1711 I0.1343 J-0.0441
N920 G02 X1.2313 Y2.1946 I0.0678 J-0.0436
N930 G02 X1.2504 Y2.1992 I0.0157 J-0.0237
N940 G02 X1.2679 Y2.1903 I-0.0034 J-0.0283
N950 G02 X1.2850 Y2.1619 I-0.0591 J-0.0548
N960 G02 X1.2924 Y2.1269 I-0.1335 J-0.0465
N970 G02 X1.2915 Y2.0812 I-0.2292 J-0.0185
N980 G02 X1.2816 Y2.0365 I-0.2283 J0.0272
N990 G02 X1.2662 Y2.0042 I-0.1343 J0.0441
N1000 G02 X1.2430 Y1.9806 I-0.0678 J0.0437
N1010 G02 X1.2239 Y1.9761 I-0.0157 J0.0237
N1020 G01 X1.2189 Y1.9768
N1030 G03 X1.1477 Y2.0069 I-1.1023 J-2.5005
N1040 G02 X1.2272 Y2.2727 I0.2132 J0.0810
N1050 G02 X1.3030 Y2.2181 I0.0154 J-0.0585
N1060 G03 X1.2028 Y2.2550 I-0.0573 J-0.0011
N1070 G03 X1.1523 Y2.0070 I0.1609 J-0.1619
N1080 G03 X1.0237 Y2.0263 I-0.1244 J-0.3915
N1090 G03 X0.9814 Y2.0450 I-0.0813 J-0.1272
N1100 G01 X0.9811 Y2.0465
N1110 G02 X0.9568 Y2.1738 I0.2169 J0.1075
N1120 G02 X1.0151 Y2.2727 I0.1375 J-0.0145
N1130 G01 X1.0283 Y2.2859
N1140 G02 X1.1040 Y2.2313 I0.0155 J-0.0583
N1150 G03 X1.0094 Y2.2736 I-0.0551 J0.0037
N1160 G01 X0.9962 Y2.2605
N1170 G03 X0.9571 Y2.1255 I0.1043 J-0.1033
N1180 G03 X0.9801 Y2.0468 I0.1949 J0.0140
N1190 G01 X0.9801 Y2.0456
N1200 G03 X0.8485 Y2.0938 I-0.3533 J-0.7601
N1210 G02 X1.1016 Y2.5166 I0.5004 J-0.0124
N1220 G02 X1.1521 Y2.4183 I-0.0167 J-0.0707
N1230 G02 X1.5536 Y2.4153 I0.1996 J-0.1490
N1240 G02 X1.5302 Y2.0909 I-0.2502 J-0.1450
N1250 G03 X1.5605 Y2.4000 I-0.2339 J0.1789
N1260 G03 X1.1515 Y2.4181 I-0.2108 J-0.1331
N1270 G03 X1.1029 Y2.5163 I-0.0684 J0.0273
N1280 G01 X1.1021 Y2.5169
N1290 G02 X1.3635 Y2.5817 I0.2467 J-0.4355
N1300 G02 X1.3860 Y3.0787 I0.1040 J0.2443
N1310 G02 X1.8971 Y3.0343 I0.1992 J-0.6707
N1320 G02 X1.7121 Y2.5271 I-0.1542 J-0.2311
N1330 G02 X1.9743 Y2.3552 I-0.0735 J-0.3981
N1340 G02 X2.6211 Y2.4181 I0.3263 J0.0020
N1350 G02 X2.6236 Y2.2065 I-0.4665 J-0.1113
N1360 G02 X2.0024 Y2.0974 I-0.3230 J0.0164
N1370 G02 X1.6211 Y1.6909 I-0.4385 J0.0292
N1380 G02 X1.6647 Y1.1627 I-0.0644 J-0.2712
N1390 G02 X1.6120 Y1.4885 I0.5694 J0.2594
N1400 G01 X1.5589 Y1.5450
N1410 X1.6127 Y1.4938
N1420 G02 X1.6211 Y1.5453 I1.3841 J-0.1985
N1430 G03 X1.8333 Y0.9454 I0.5996 J-0.1254
N1440 G01 X1.8181 Y0.9272
N1450 G03 X2.7987 Y0.8426 I0.5898 J1.1113
N1460 G02 X2.9131 Y0.6380 I0.0565 J-0.1027
N1470 G02 X2.7401 Y0.6673 I-0.0680 J0.1240
N1480 G03 X2.8872 Y0.6599 I0.0792 J0.1079
N1490 G03 X2.8333 Y0.7999 I-0.0271 J0.0700
N1500 G02 X1.7727 Y0.8545 I-0.4590 J1.4119
N1510 G01 X1.7424 Y0.8363
N1520 G03 X2.0302 Y0.6181 I0.3614 J0.1780
N1530 G02 X2.1186 Y0.4948 I0.0453 J-0.0609
N1540 G02 X2.4323 Y0.3814 I0.1064 J-0.1962
N1550 G02 X2.4172 Y0.2716 I-0.1251 J-0.0389
N1560 G02 X2.1494 Y0.0904 I-0.3462 J0.2232
N1570 G02 X1.7272 Y0.1454 I-0.1355 J0.6075
N1580 G02 X1.8181 Y0.4181 I0.1290 J0.1085
N1590 G02 X1.7727 Y0.5454 I-0.0238 J0.0632
N1600 G03 X1.5454 Y0.7272 I-0.3371 J-0.1885
N1610 G01 X1.4241 Y0.7454
N1620 G03 X1.1818 Y0.8908 I-0.4466 J-0.4697
N1630 G02 X1.4241 Y0.7454 I-0.2043 J-0.6151
N1640 G01 X1.5454 Y0.7272
N1650 G02 X1.7727 Y0.5454 I-0.1098 J-0.3703
N1660 G03 X1.8181 Y0.4181 I0.0215 J-0.0641
N1670 G03 X1.7272 Y0.1454 I0.0381 J-0.1642
N1680 G02 X1.1263 Y0.0937 I-0.3440 J0.4804
N1690 G02 X1.0841 Y0.3102 I0.0739 J0.1267
N1700 G02 X1.5302 Y0.4362 I0.3070 J-0.2341
N1710 G02 X1.6211 Y0.5272 I0.0545 J0.0364
N1720 G03 X1.3333 Y0.7272 I-0.5648 J-0.5057
N1730 G02 X1.1216 Y0.7453 I-0.0454 J0.7133
N1740 G01 X1.1191 Y0.7453
N1750 X1.0817 Y0.7464
N1760 X0.7592 Y0.7470
N1770 M00
N1780 M02
N1790 M30
```

### Package Logical/Libraries - Globale Bibliotheken

- Visualisation Logical/Visualization (not shown)

Listed in the project but not available here: Logical/Global.typ, Logical/Global.var, Logical/Motion/Cnc/ActionMpLogging.st, Logical/Motion/MFunc/Exit.st, Logical/Motion/MFunc/Types.typ, Logical/Motion/acp10etxen, Logical/GmcIpConfig/gmcipsys, Logical/GmcIpConfig/gmciplbr, Logical/GmcIpConfig/gmcipcbr, Logical/GmcIpConfig/gmciplsm, Logical/GmcIpConfig/gmcipcsm, Logical/GmcIpConfig/gmcipcfg, Logical/GmcIpConfig/gmcipiec, Logical/GmcIpConfig/gmciplog, Logical/GmcIpConfig/gmcipesm, Logical/GmcIpConfig/gmcipmxd, Logical/GmcIpConfig/gmcipmx, Logical/GmcIpUserConfig/gmcipvar, Logical/GmcIpUserConfig/gmcipfun, Logical/GmcIpUserConfig/gmcipfub, Logical/GmcIpUserConfig/gmcipubr, Logical/GmcIpUserConfig/gmcipusm, Logical/GmcIpUserConfig/gmcipui, Logical/GmcIpUserConfig/gmcipus, Logical/GmcIpUserConfig/gmcipuc
